// TIA Portal V17 export
// export: Created 2025-03-05T08:00:31.890285Z, ExportSetting WithDefaults, DisplayName Totally Integrated Automation Portal, DisplayVersion V17 Update 8, DisplayName TIA Portal Openness, DisplayVersion V17 Update 8, DisplayName TIA Portal Version Control Interface, DisplayVersion V17, DisplayName SINAMICS Startdrive Advanced, DisplayVersion V17 SP2, DisplayName SINAMICS Startdrive G110M, G120, G120C, G120D, G120P, G115D, DisplayVersion V17 SP2, DisplayName SINAMICS Startdrive G130, G150, S120, S150, SINAMICS MV, S210, DisplayVersion V17 SP2, DisplayName STEP 7 Professional, DisplayVersion V17 Update 8, DisplayName SINUMERIK ONE STEP 7 Toolbox, DisplayVersion V17 Update 12, DisplayName SINUMERIK 840D sl STEP 7 Toolbox, DisplayVersion V17 Update 12, DisplayName STEP 7 Safety, DisplayVersion V17 Update 6, DisplayName WinCC Advanced, DisplayVersion V17 Update 8
DATA_BLOCK "DB1231_UNIT_01_PART_CHECK_STATION_0"   // DB1231
{ S7_Optimized_Access := 'FALSE'; DB_Accessible_From_OPC_UA := 'FALSE' }
VERSION : 0.1
// stored: AutoNumber false, DBAccessibleFromOPCUA false, DBAccessibleFromWebserver true, IsOnlyStoredInLoadMemory false, IsWriteProtectedInAS false
   VAR
      SEQUENCE : "RUN_CNC_SEQ";
      ANY_DOOR_OPEN_MEM { S7_SetPoint := 'True'} : Bool;   // ANY DOOR OPEN MEMORY
      FIX_1_CLAMP_LOST_MEM : Bool;   // FIXTURE 1 CLAMP LOST MEMORY
      FIX_2_CLAMP_LOST_MEM : Bool;   // FIXTURE 2 CLAMP LOST MEMORY
      FIX_3_CLAMP_LOST_MEM : Bool;   // FIXTURE 3 CLAMP LOST MEMORY
      FIX_4_CLAMP_LOST_MEM : Bool;   // FIXTURE 4 CLAMP LOST MEMORY
      AUX_PULSE_1 : Bool;
      AUX_PULSE_2 : Bool;   // AUX PULSE 1
      AUX_PULSE_3 : Bool;   // AUX PULSE 1
      AUX_PULSE_4 : Bool;   // AUX PULSE 1
      AUX_PULSE_5 : Bool;   // AUX PULSE 1
   END_VAR
BEGIN
   SEQUENCE.TIMER_TIME_EXCEED.PT := T#2M;
END_DATA_BLOCK
